RoboDK station: WartenDI.rdk

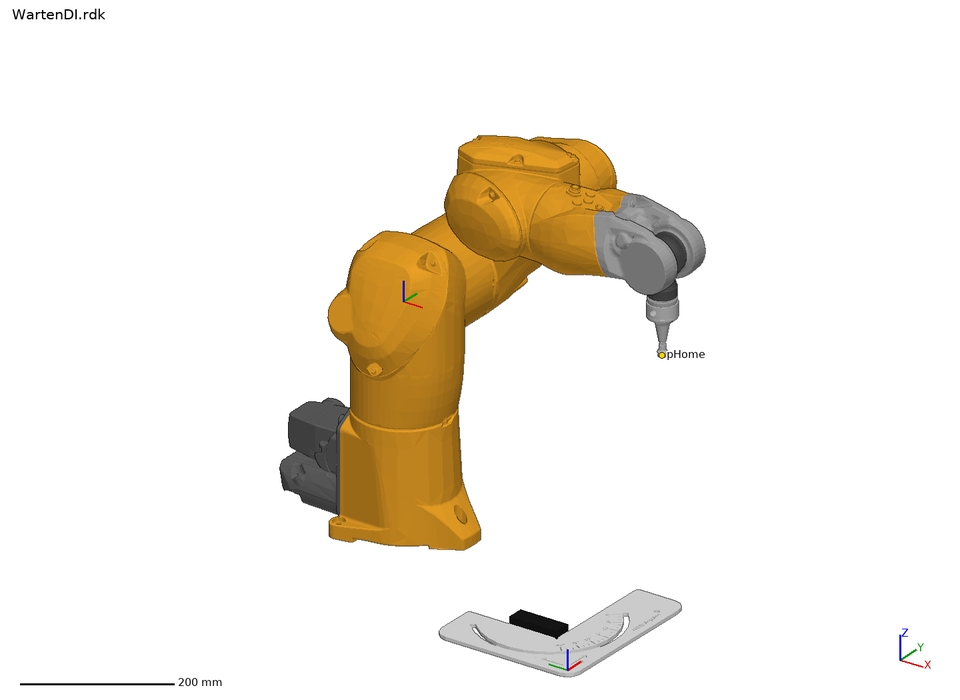
[picture v0: the station drawn from its stored meshes, robots at their saved joint values, targets as dots, program paths as lines]
Station WartenDI (saved by RoboDK 5.0.2). Poses are relative to the parent item; angles as X-Y-Z fixed-axis rotations.
Station parameters (name, value as stored): Vacuum, 1
  - frame world at (0, 0, 0) mm
    - frame Staubli TX2-40 Base at (0, 0, 0) mm
      - robot Staubli TX2-40: 6 axes, payload 1.7 kg, reach 515 mm, repeatability 0.02 mm, weight 29 kg
          modified DH rows (alpha deg, a mm, theta deg, d mm): 0, 0, 0, 320; -90, 0, -90, 35; 0, 225, -90, 0; -90, 0, 0, 225; 90, 0, 0, 0; -90, 0, 180, 65
          base shift (0, 0, -320) mm
          joint limits [-180, -125, -138, -190, -120, -270] to [180, 125, 138, 190, 133.5, 270]; home [0, 0, 90, 0, 0, 0]; saved at [0, 45, 45, 0, 90, 0]
        - tool LWS_VakuumGreifer_14, TCP at (0, 0, 78) mm, size 81.8 x 45.9 x 42 mm, geometry from LWS_VakuumGreifer_14.stl
      - target pHome (joint target) at (384.1, 35, 16.1) mm, rotated rx 180 ry 0 rz -180 deg; joints [0, 45, 45, 0, 90, 0] of Staubli TX2-40
      - frame MagazineFrame at (399.83, -201.23, -338.58) mm, rotated rx 0 ry 0 rz 89.57 deg
        - object Schlosserwinkel_AROB at (0, 0, 0) mm, size 260 x 220 x 5 mm, geometry from Schlosserwinkel_AROB.stp
  - Python program WartenDI (listed below)
  - object Jengastuck 1 at (302.39, -127.49, -323.58) mm, rotated rx 0 ry 0 rz 89.57 deg, size 75 x 25 x 15 mm, geometry from Jengastuck.stp

--- Python program WartenDI ---
# BEISPIELPROGRAMM: RTS-LIBRARY: WARTEN AUF DIGITALEN EINGANG
# Führt 2 Bewegungen aus und gibt dann eine Nachricht einerseits
# in der Simulation, und andererseits auf dem Robotercontroller aus.

# Import der Librarys
from robolink import *
from robodk import *
from RTS import *

RDK = Robolink()

# Initialisierung aller Simulationsobjekte
r_tx240 = RDK.Item("Staubli TX2-40", ITEM_TYPE_ROBOT)
g_gripper = RDK.Item("LWS_VakuumGreifer_14")
f_magazine = RDK.Item("MagazineFrame", ITEM_TYPE_FRAME)
f_world = RDK.Item("world", ITEM_TYPE_FRAME)
f_robot = RDK.Item("Staubli TX2-40 Base", ITEM_TYPE_FRAME)
pHome = RDK.Item("pHome", ITEM_TYPE_TARGET)
block = RDK.Item("Jengastuck 1")

# Erstellen des RTS-Objektes.
RTS = RTS(RDK, r_tx240, g_gripper)

# Initialisieren der Verbindung des Vakuumgreifers.
RTS.addConnection("dVacuum","98FE10BA-0446-4B8A-A8CF-35B98F42725A","dio")

# Initialisieren der Verbindung des Vakuumsensors.
RTS.addConnection("dVacuumSensor","BFFF5B02-EDA8-4EAA-AB65-0D4DAB2D24C5","dio")

# Setzen der Verbindung dVacuum als Greifer des Roboters.
RTS.setGripperConnection("dVacuum")

# Berechnung und Bewegung zu den Punkten.
IntermediatePose = transl(254, -30, -190) * rotx(-pi) * rotz(pi)

r_tx240.MoveJ(pHome)
r_tx240.MoveJ(IntermediatePose)

BlockPosition = block.PoseAbs()
PickUpPosition = BlockPosition
PickUpPosition = PickUpPosition * rotx(-pi) * rotz(-pi/2)

PickApproachPosition= PickUpPosition * rotz(2*pi)
PickApproachPosition=PickApproachPosition * transl(0, 0, -50)

r_tx240.MoveJ(PickApproachPosition)
r_tx240.MoveL(PickUpPosition)

# Setzen des Vakuums. Setzt dies in der Simulation und
# auf dem Roboter (Insofern der Greifer richtig initialisiert wurden.)
RTS.setVacuum(1)

# Wartet, bis der Eingang dVacuumSensor 1 ist, oder das Timeout von 5 Sekunden abgelaufen ist.
# Hat keinen Einfluss auf die Simulation.
RTS.waitConnection("dVacuumSensor", 1, 5)

# Bewegt Roboter zu folgenden 4 Punkten, unabhängig davon, ob ein Vakuum gefunden wurde oder nicht.
r_tx240.MoveL(PickApproachPosition)
r_tx240.MoveJ(IntermediatePose)
r_tx240.MoveJ(PickApproachPosition)
r_tx240.MoveL(PickUpPosition)

# Lässt den Block wieder los.
RTS.setVacuum(0)
r_tx240.MoveJ(pHome)
